{attribute 'OPC.UA.DA' := '1'}
FUNCTION_BLOCK PsdChamber EXTENDS ChamberBase
VAR_INPUT
	IoChamberPsd : IoChamberPsd;	
END_VAR
VAR_OUTPUT
END_VAR
VAR
	{attribute 'OPC.UA.DA' := '0'}
	_config : PsdChamberConfig;
	
	{attribute 'OPC.UA.DA' := '0'}
	_initDevice : BOOL;
	
	{attribute 'OPC.UA.DA' := '0'}
	_itemInit : INT;
	{attribute 'OPC.UA.DA' := '0'}
	_itemScheduler : INT;
	{attribute 'OPC.UA.DA' := '0'}
	_itemExecScheduler : INT;		
	{attribute 'OPC.UA.DA' := '0'}
	_itemRaisedProperties : INT;			
	{attribute 'OPC.UA.DA' := '0'}
	_pulseGenerator : TON;	
	
	{region 'Commands'}	
		 	
	{attribute 'OPC.UA.DA' := '0'}
	_enableCamera : BOOL;
	{attribute 'OPC.UA.DA' := '0'}
	_moveSlitDoorPositionCmd : BOOL;
	{attribute 'OPC.UA.DA' := '0'}
	_moveCdaPneumaticValveCmd : BOOL;
	{attribute 'OPC.UA.DA' := '0'}			  		   
	_raisePropertiesCmd : BOOL;	 
			
	{endregion}
	
	{attribute 'OPC.UA.DA' := '0'}
	_deliverMessages : INT;
	
	InterlockPanelsMsg : STRING(255);	
	SlitDoorPositionMsg : STRING(255);	
	SlitDoorOpenPositionMsg : STRING(255);
	SlitDoorClosePositionMsg : STRING(255);
	CdaValveIsOpenMsg : STRING(255);
	RefreshingMsg : STRING(255);
		
	{attribute 'OPC.UA.DA' := '0'}
	message : STRING(255);
	
	{attribute 'OPC.UA.DA' := '0'}
	_pos : INT;
	{attribute 'OPC.UA.DA' := '0'}
	_openCdaValve : BOOL;
	{attribute 'OPC.UA.DA' := '0'}
	_cdaValveIsOpen : BOOL;
	
	
	{attribute 'OPC.UA.DA' := '0'}
	tmpConcat1 : STRING;
	{attribute 'OPC.UA.DA' := '0'}
	tmpConcat2 : STRING;
	{attribute 'OPC.UA.DA' := '0'}
	tmpConcatName : STRING; 
	{attribute 'OPC.UA.DA' := '0'}
	tmpConcatDescription : STRING;
	{attribute 'OPC.UA.DA' := '0'}
	tmpConcatInterlockID : STRING;
	
	{attribute 'OPC.UA.DA' := '0'}
	_itemInterlock : UINT;
	{attribute 'OPC.UA.DA' := '0'}
	_interlockCount : UINT;
		
END_VAR

SUPER^();
 
// Init device
InitDevice(); 

// Deliver messages
CASE _deliverMessages OF	
	EFeedbackMsgPsdChamber.InterlockPanelsMsg :
		InterlockPanelsMsg := message;	
	EFeedbackMsgPsdChamber.SlitDoorPositionMsg :
		SlitDoorPositionMsg := TO_STRING(SlitDoorPosition);
	EFeedbackMsgPsdChamber.SlitDoorOpenPositionMsg :
		SlitDoorOpenPositionMsg := TO_STRING(SlitDoorOpenPosition);
	EFeedbackMsgPsdChamber.SlitDoorClosePositionMsg :
		SlitDoorClosePositionMsg := TO_STRING(SlitDoorClosePosition);
	EFeedbackMsgPsdChamber.CdaValveIsOpenMsg :
		CdaValveIsOpenMsg := TO_STRING(_cdaValveIsOpen);	
END_CASE

// Commands
MoveSlitDoorPosition(_moveSlitDoorPositionCmd, _pos); 
MoveCdaPneumaticValve(_moveCdaPneumaticValveCmd, _openCdaValve); 
RaisePropertiesChanged(_raisePropertiesCmd);

IF NOT _moveSlitDoorPositionCmd AND NOT _raisePropertiesCmd THEN	
	MessageScheduler();
END_IF

PROPERTY CdaValveIsOpen : BOOL
GET
CdaValveIsOpen := _cdaValveIsOpen;
END_GET
SET
_cdaValveIsOpen := CdaValveIsOpen;
END_SET
END_PROPERTY

METHOD FB_init : BOOL
VAR_INPUT
	bInitRetains : BOOL; // if TRUE, the retain variables are initialized (warm start / cold start)
	bInCopyCode : BOOL;  // if TRUE, the instance afterwards gets moved into the copy code (online change)
	Config : PsdChamberConfig;
END_VAR
IF Config.IsEnabled THEN
	_config := Config;
	
	SUPER^._chamberConfig.Name := Config.Name;
	SUPER^._chamberConfig.DeviceID := Config.DeviceID;
	SUPER^._chamberConfig.IsEnabled := Config.IsEnabled;
	SUPER^._chamberConfig.LogLevel := Config.LogLevel;
	
	SUPER^.Name := Config.Name;
	SUPER^.DeviceID := Config.DeviceID;
	
	THIS^.Family := DeviceFamily.Chamber;

	THIS^.SetReady();
	_Logger.Information(_message.Reset().Append('Init ').
							Append('{').Append(TO_STRING(THIS^.Family)).Append('} - ').
							Append('{').Append(TO_STRING(THIS^.Name)).Append('} - ').
							Append('Status : ').Append(TO_STRING(THIS^.Status)).
							ToString());										 
END_IF
END_METHOD

METHOD InitDevice
VAR_INPUT
END_VAR
VAR	
END_VAR
IF NOT _initDevice THEN			
	_logger.Information(_message.Reset().
								Append(_config.Name).
								Append(' - init device').ToString());		
								
	IF IoChamberPsd.OutputCdaPneumaticValve = FALSE THEN
		_logger.Information(_message.Reset().Append('Start pneumatic valve').ToString());								
		IoChamberPsd.OutputCdaPneumaticValve := TRUE;
	END_IF
	
	_initDevice := TRUE;
END_IF
END_METHOD

METHOD MessageScheduler
VAR_INPUT
END_VAR
IF _pulseGenerator.Q THEN
	_pulseGenerator(IN := FALSE, PT := T#10MS);
		
	CASE _itemScheduler OF	
		0: SlitDoorPositionMsg := ' ';		   
		   CdaValveIsOpenMsg := ' ';
		   _itemScheduler := 1;
		   
		1: ReadInterlock();
		   _itemScheduler := 2;
		   
		2:  ReadSlitDoorPosition();
			_itemScheduler := 3;

		3:  ReadSlitDoorOpenPosition();
			_itemScheduler := 4;

		4:  ReadSlitDoorClosePosition();
			_itemScheduler := 5;		
					
		5:  IsReadyToLoadUnload();
			_itemScheduler := 6;	
		
		6:  ReadCdaValvePosition();
			_itemScheduler := 0;					
	END_CASE
ELSE
	_pulseGenerator(IN := TRUE, PT := T#50MS);		
END_IF
END_METHOD

{attribute 'TcRpcEnable' := '1'}
METHOD MoveCdaPneumaticValve
VAR_INPUT
	Execute : BOOL;
	OpenValve : BOOL;
END_VAR
IF Execute THEN
	_logger.Information(_message.Reset().Append(_config.Name).Append(' - Move CDA pneumatic valve : ').Append(TO_STRING(openValve)).ToString());
		
	IF OpenValve THEN
		IoChamberPsd.OutputCdaPneumaticValve := TRUE;
	ELSE
		IoChamberPsd.OutputCdaPneumaticValve := FALSE;	
	END_IF			
	
	_openCdaValve := FALSE;
END_IF
END_METHOD

{attribute 'TcRpcEnable' := '1'}
METHOD MoveSlitDoorPosition
VAR_INPUT
	Execute : BOOL;
	Position : INT;
END_VAR
IF Execute THEN
	_logger.Information(_message.Reset().Append(_config.Name).Append(' - Move slit door position : ').Append(TO_STRING(Position)).ToString());
	
	_moveSlitDoorPositionCmd := FALSE;
	
	IF Position = ESlitDoorPosition.Open THEN
		IoChamberPsd.OutputOpenSlitDoor := TRUE;
		IoChamberPsd.OutputCloseSlitDoor := FALSE;
	ELSIF Position = ESlitDoorPosition.Close THEN
		IoChamberPsd.OutputOpenSlitDoor := FALSE;
		IoChamberPsd.OutputCloseSlitDoor := TRUE;
	ELSE
		_logger.Error(_message.Reset().Append(_config.Name).Append(' - unknown position : ').Append(TO_STRING(Position)).ToString());
	END_IF
			
	_itemScheduler := 0;
END_IF
END_METHOD

{attribute 'TcRpcEnable' := '1'}
METHOD RaisePropertiesChanged
VAR_INPUT
	Execute : BOOL;
END_VAR
IF Execute THEN		
	_raisePropertiesCmd := TRUE;	
		
	IF _pulseGenerator.Q THEN
		_pulseGenerator(IN := FALSE, PT := T#10MS);
		
		CASE _itemRaisedProperties OF		
			0: 	SUPER^._raisePropertiesBase := TRUE;	
				RefreshingMsg := TO_STRING(TRUE);
				SlitDoorPositionMsg := TO_STRING(ESlitDoorPosition.Unknown);				   
				_itemRaisedProperties := 1;
			
			1:  SlitDoorOpenPositionMsg := ' ';
				_itemRaisedProperties := 2;
				
			2:	SlitDoorClosePositionMsg := ' ';
				_itemRaisedProperties := 3;
				
			3:  CdaValveIsOpenMsg := ' ';	   
				_itemRaisedProperties := 4;
				
			4:  ReadInterlock();
				_itemRaisedProperties := 5;
				
			5:  ReadInterlock();
				_itemRaisedProperties := 6;
				
			6:  ReadInterlock();
				_itemRaisedProperties := 7;
				
			7:  ReadInterlock();
				_itemRaisedProperties := 8;
				
			8:  ReadInterlock();
				_itemRaisedProperties := 9;
				
			9:  ReadInterlock();
				_itemRaisedProperties := 10;						
				
			10: RefreshingMsg := TO_STRING(FALSE);
				_itemRaisedProperties := 20;
				
			20: _logger.Information(_message.Reset().Append(_config.Name).Append(' - RaisePropertiesChanged').ToString());
				_raisePropertiesCmd := FALSE;
				_itemRaisedProperties := 0;
		END_CASE	
	ELSE
		_pulseGenerator(IN := TRUE, PT := T#100MS);	
	END_IF		
END_IF
END_METHOD

METHOD ReadCdaValvePosition 
VAR_INPUT
END_VAR
VAR
END_VAR
_deliverMessages := EFeedbackMsgPsdChamber.CdaValveIsOpenMsg;


IF IoChamberPsd.OutputCdaPneumaticValve THEN
	CdaValveIsOpen := TRUE;
ELSE
	CdaValveIsOpen := FALSE;	
END_IF
END_METHOD

METHOD ReadInterlock 
VAR_INPUT
END_VAR
VAR
	statePanel : STRING;
END_VAR
_deliverMessages := EFeedbackMsgPsdChamber.InterlockPanelsMsg;

IF _interlockCount < Const.PSD_NUMBER_INTERLOCK_PANELS THEN
	_interlockCount := _interlockCount + 1;
ELSE
	_interlockCount := 0;
END_IF

tmpConcatName := CONCAT(_config.Interlock[_interlockCount].Name, ';');
tmpConcatDescription := CONCAT(_config.Interlock[_interlockCount].Description, ';');
tmpConcatInterlockID := CONCAT(UINT_TO_STRING(_config.Interlock[_interlockCount].InterlockID), ';');

tmpConcat1 := CONCAT(tmpConcatName, tmpConcatDescription);
tmpConcat2 := CONCAT(tmpConcat1, tmpConcatInterlockID);

IF _config.Interlock[_interlockCount].State THEN
	statePanel := 'Closed';
ELSE
	statePanel := 'Open';
END_IF

message := CONCAT(tmpConcat2, statePanel);
END_METHOD

METHOD ReadSlitDoorClosePosition 
VAR_INPUT
END_VAR
VAR
	open : BOOL;
	close : BOOL;
END_VAR
_deliverMessages := EFeedbackMsgPsdChamber.SlitDoorClosePositionMsg;
SlitDoorClosePosition := IoChamberPsd.InputCloseSlitDoor;
END_METHOD

METHOD ReadSlitDoorOpenPosition 
VAR_INPUT
END_VAR
VAR
END_VAR
_deliverMessages := EFeedbackMsgPsdChamber.SlitDoorOpenPositionMsg;
SlitDoorOpenPosition := IoChamberPsd.InputOpenSlitDoor;
END_METHOD

METHOD ReadSlitDoorPosition 
VAR_INPUT
END_VAR
VAR
	open : BOOL;
	close : BOOL;
	efemOpen : BOOL;
END_VAR
_deliverMessages := EFeedbackMsgPsdChamber.SlitDoorPositionMsg;

open := IoChamberPsd.InputOpenSlitDoor;
close := IoChamberPsd.InputCloseSlitDoor;
efemOpen := IoChamberBase.InputEfemSlitDoorOpen;

IF open AND NOT close AND efemOpen THEN
	SlitDoorPosition := ESlitDoorPosition.Open;	
ELSIF close AND NOT open AND NOT efemOpen THEN
	SlitDoorPosition := ESlitDoorPosition.Close;
ELSIF close AND open THEN
	SlitDoorPosition := ESlitDoorPosition.Error;	
ELSE
	SlitDoorPosition := ESlitDoorPosition.Unknown;		
END_IF
END_METHOD

END_FUNCTION_BLOCK

(* stored: Version 1.1.0.1, ProductVersion 3.1.4024.12
   POU PsdChamber: Id {5cb78e1f-1a67-4eed-b24c-c353ece2e6da}, SpecialFunc None
   Folder Commands: Id {446636a9-e1bf-41a2-beda-5f71ee3f8bbe}
   Property CdaValveIsOpen: Id {fbc715b0-8664-4d4b-a96c-4aeb352ceedd}
   Get Get: Id {1fb41dee-8162-494f-b169-40ee8f0fcd2b}
   Set Set: Id {b9fa4638-3401-46bd-8111-5363d90470b8}
   Method FB_init: Id {19c0411c-4163-4a09-896a-4fc7f328f179}
   Method InitDevice: Id {77f938ff-dece-4e7c-a91b-89fd1a1b8513}
   Method MessageScheduler: Id {b363294c-b909-46ca-a08f-67a2fb547bf6}
   Method MoveCdaPneumaticValve: Id {83961ea3-238a-48de-90d5-24ef42374b79}
   Method MoveSlitDoorPosition: Id {9467c568-9014-4226-9d21-944c103d853b}
   Method RaisePropertiesChanged: Id {83701a8c-91db-4288-a78c-d25d8d620e09}
   Method ReadCdaValvePosition: Id {e818dd7c-bee3-4da3-ae75-6cc8ead65710}
   Method ReadInterlock: Id {37993eea-98d8-4d0e-b584-e5891f3e239d}
   Method ReadSlitDoorClosePosition: Id {5473a5f3-41d4-4dc8-9db3-035535aff6f4}
   Method ReadSlitDoorOpenPosition: Id {55623f1f-95a6-4e5e-a4ab-86cb74e27085}
   Method ReadSlitDoorPosition: Id {d0053aee-5cad-4557-8192-2b2532ce0e65} *)
